TEXTLIST TextListForCombobox_eReglertyp
  1 = 'P'
  2 = 'I'
  3 = 'PI'
  4 = 'PDT1'
  5 = 'PIDT1'
   = ''
END_TEXTLIST

(* stored: Version 1.1.0.1, ProductVersion 3.1.4024.12
   TextList TextListForCombobox_eReglertyp: Id {5575e17a-6d73-4d4f-95de-15ded094f467} *)
